Yaskawa INFORM job: _DEL13.JBI

/JOB
//NAME _DEL13
//POS
///NPOS 0,0,0,0,0,0
//INST
///DATE 2018/08/28 16:52
///ATTR SC,RW,MC
NOP
END
